TYPE (* Value of auxiliary inputs Struct *)
  (* Version 1.0, 2025-07-21, franz *)
  PACKAGE isobus::UT_io::aux::in;
  AuxiliaryState_S : STRUCT
    value : USINT := 255;
    bCyclic : BOOL := TRUE; (* do not repeat every 200ms if this is set FALSE *)
  END_STRUCT;
END_TYPE
